FUNCTION_BLOCK FB_TimedButton
VAR_INPUT
	bIsTimeButtonPressed : BOOL;
	tMaxTime : TIME;	// Maximum time to hold the button before swithing lights
END_VAR
VAR_OUTPUT
	bLightOfTimedButton : BOOL;
	bLightOfOtherButton : BOOL;
END_VAR
VAR
	fbTimerForTimedButton : TON;	// For timing the button press
	tTimePressed : DWORD;
	
	sMaxTime : DWORD := 3000;
END_VAR

IF bIsTimeButtonPressed  THEN	// Check if the time button is pressed
	tMaxTime := DWORD_TO_TIME(sMaxTime);
	fbTimerForTimedButton(IN := TRUE, PT := tMaxTime);	// Start the timer
	tTimePressed := TIME_TO_DWORD(fbTimerForTimedButton.ET);
	// If timer hasn't reached max time, turn on first light, ensure second light is off
	IF NOT fbTimerForTimedButton.Q THEN
		bLightOfTimedButton := TRUE;
		bLightOfOtherButton := FALSE;
	// If timer has reached max time, turn off first light, turn on second light
	ELSE
		bLightOfTimedButton := FALSE;
		bLightOfOtherButton := TRUE;
	END_IF
ELSE	// Button is not pressed
	fbTimerForTimedButton(IN := FALSE);	// Reset the timer
	// Both lights should be off
	bLightOfTimedButton := FALSE;
	bLightOfOtherButton := FALSE;
END_IF

END_FUNCTION_BLOCK

(* stored: Version 1.1.0.1, ProductVersion 3.1.4024.12
   POU FB_TimedButton: Id {1061c217-a255-481c-86c6-ed62e22d1040}, SpecialFunc None *)
